# EPICS autosave request: iocBoot/ioc13Syringe2/auto_settings.req
file "CPSyringe_settings.req",         P=$(P), R=$(R)
